{attribute 'qualified_only'}
{attribute 'strict'}
TYPE eTcoMultiAxisSystem :
(
	SingleAxisSystem := 1,
	TwoAxisSystem := 2,
	ThreeAxisSystem := 3,
	FourAxissystem := 4

);
END_TYPE

(* stored: Version 1.1.0.1, ProductVersion 3.1.4024.12
   DUT eTcoMultiAxisSystem: Id {c90cee85-4ef5-06ca-3149-7bb41bf7d22c} *)
